(* PLC project OOP_Curso, Beckhoff Automation GmbH TwinCAT PLC Control 3.5.13.21 *)
(* stored: creationDateTime 2023-10-22T17:41:31.5511473, modificationDateTime 2023-10-22T17:41:31.557005 *)

INTERFACE I_Humano
METHOD Correr
VAR_INPUT
END_VAR
END_METHOD
PROPERTY Nombre : STRING
END_PROPERTY
END_INTERFACE

FUNCTION_BLOCK Corazon
VAR_INPUT
END_VAR
VAR_OUTPUT
END_VAR
VAR
	VarHumano: Humano;
	pHumano: POINTER TO Humano;
	pHumano16: REFERENCE TO Humano;
END_VAR

            
          
END_FUNCTION_BLOCK

FUNCTION_BLOCK Hombre EXTENDS Humano
VAR_INPUT
END_VAR
VAR_OUTPUT
END_VAR
VAR
END_VAR

            
          
END_FUNCTION_BLOCK

FUNCTION_BLOCK Humano IMPLEMENTS I_Humano
VAR_INPUT
END_VAR
VAR_OUTPUT
END_VAR
VAR
END_VAR

            
          

{warning 'Agregar implementación de método'}
METHOD Correr
                  
                
END_METHOD

{warning 'Agregar implementación de propiedad'}
PROPERTY Nombre : STRING
GET
VAR
END_VAR
                    
                  
END_GET
SET
VAR
END_VAR
                    
                  
END_SET
END_PROPERTY
END_FUNCTION_BLOCK

FUNCTION_BLOCK Sangre
VAR_INPUT
END_VAR
VAR_OUTPUT
END_VAR
VAR
	VarHumano: Humano;
END_VAR

            
          
END_FUNCTION_BLOCK
